Fanuc KAREL source: kt00453.KL

-- PROVISIONAL review KL for V770-1; original PC SHA256 906c4b389afb14cdea834c3d98a67f917e9ef64545ce4fbd2f31dce9b8241bb2
-- Incomplete behavior may be omitted. Consult companion uncertainty JSON. Do not deploy.
PROGRAM KT00453
%NOLOCKGROUP
VAR
  OUT : BOOLEAN
-- UNRESOLVED_DECL H1 type=002017
-- UNRESOLVED_DECL Y2 type=002018
BEGIN
  -- UNRESOLVED_PC offsets 5-19; opcodes 2E,22,9D,33,B4
  -- UNRESOLVED_PC offsets 24-38; opcodes 2E,22,9D,33,B2
  -- UNRESOLVED_PC offsets 43-68; opcodes 22,9D,33,B3,22,9D,33,B1,5C,23
  -- UNRESOLVED_PC offsets 73-77; opcodes 7F
END KT00453
